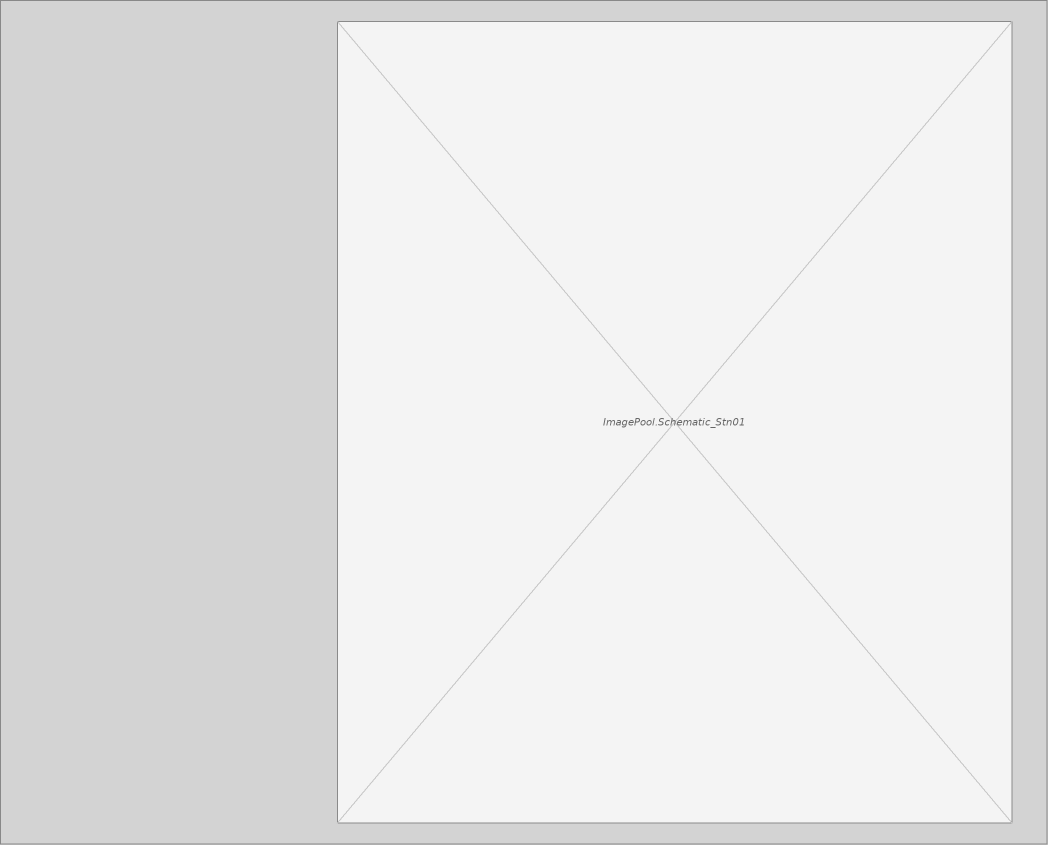
VISUALIZATION Recipe_Station11  // 1048x845
    Rectangle (0,0 1048x845)
    Image (337,21 675x802), image: ImagePool.Schematic_Stn01
END_VISUALIZATION

(* stored: Version 1.1.0.1, ProductVersion 3.1.4024.12
   Visu Recipe_Station11: Id {1539f68d-7461-4108-8314-b30c219e2b35} *)
